(* CoDeSys 2.3 export: ADS_COMMUNICATION.EXP *)

(* POU ADS_Communication, CFC *)
PROGRAM ADS_Communication
VAR
	fb_floor3ADSwrite: ADSWRITE;


	counter_error,counter_busy: CTU;
END_VAR
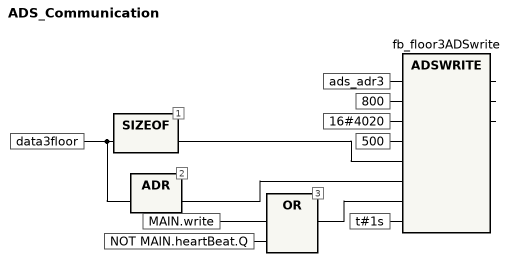
_CFC_ (* Continuous Function Chart, elements in execution order *)
#0 fb_floor3ADSwrite:ADSWRITE(ads_adr3, 800, 16#4020, 500, #1, #2, #3, t#1s)
#1 SIZEOF(data3floor)
#2 ADR(data3floor)
#3 OR(MAIN.write, NOT MAIN.heartBeat.Q)
_END_CFC_
END_PROGRAM
